PROGRAM MockServer
VAR
	//Mock Server
	fbhttpClient : FB_IotHttpClient := (sHostName:='4446f140-18dd-4b14-8279-3cc341a02b1e.mock.pstmn.io',
								  	bKeepAlive:=TRUE, tConnectionTimeout:=T#10S);		
				
	//Get Request
	fbRequest : FB_IotHttpRequest;		
	state : (IDLE, SEND_REQUEST, WAIT_FOR_RESPONSE, READ_RESPONSE,ERROR,HEADER);			
	sendGetRequest: BOOL;
	debugContent : STRING(511);
	fbJsonParser : FB_JsonDomParser;
	jsonDoc				: SJsonValue;
	jsonArgsMember				: SJsonValue;
	jsonMachineName : SJsonValue;
	results : STRING;
	
	//Header
	fbHeaderField : FB_IotHttpHeaderFieldMap;
END_VAR

// Init client parameters at startup
IF NOT fbhttpClient.bConfigured THEN 
	fbhttpClient.nHostPort:= 443; //80 for http  443 For https
	fbhttpClient.stTLS.bNoServerCertCheck:= TRUE;
END_IF

	
//Get Request
CASE state OF
	
	//Send Get Request
	IDLE:
		IF sendGetRequest THEN
			state := HEADER;
			sendGetRequest := FALSE;
		END_IF
	
	//Create Autorization Header File
	HEADER:
		fbHeaderField.AddField(sField:='Header1',sValue:='1',bAppendValue:=FALSE);
		fbHeaderField.AddField(sField:='Header2',sValue:='2',bAppendValue:=FALSE);
		state := SEND_REQUEST;
	
	//Send Get Request
	SEND_REQUEST:                                                                                      
		IF fbRequest.SendRequest(sUri:='/getmockdata', 
			fbClient:=fbhttpClient, eRequestType:=ETcIotHttpRequestType.HTTP_Get, 
				0, 0,fbHeader:=fbHeaderField ) THEN
			state := WAIT_FOR_RESPONSE;
		END_IF
	
	//Wait for Response
	WAIT_FOR_RESPONSE:

		IF NOT fbRequest.bBusy THEN
			IF fbRequest.bError THEN
				state := ERROR;
			ELSE
				state := READ_RESPONSE;
			END_IF
		END_IF
	
	//Read Response	
	READ_RESPONSE:
	
		//Get Response Content
		fbRequest.GetContent(pContent:= ADR(debugContent), nContentSize:= SIZEOF(debugContent), bSetNullTermination:= TRUE);
		
		//Check Status 
		IF fbRequest.nStatusCode >= 200 AND fbRequest.nStatusCode < 300 THEN
			jsonDoc:= fbRequest.GetJsonDomContent(fbJsonParser);
			
			//Check response has data in body
			IF jsonDoc <> 0 THEN
				
				//Check machine key is present 
				IF fbJsonParser.HasMember(jsonDoc, 'machine') THEN
					
					//Get Value for the specifed key
					jsonArgsMember:= fbJsonParser.FindMember(jsonDoc, 'machine');
					
					//Check wether data has an name key 	
					IF fbJsonParser.HasMember(jsonArgsMember, 'name')  THEN
						
						//Get Value for the specifed key
						jsonMachineName:= fbJsonParser.FindMember(jsonArgsMember, 'name');
						
							//Check data is a String
							IF fbJsonParser.IsString(jsonMachineName) THEN	
								
								//Get the Data 		
								results:= fbJsonParser.GetString(jsonMachineName);									
							END_IF
					END_IF
				END_IF
			END_IF
		END_IF
		state := IDLE;
		
	ERROR:
		//
		
		
END_CASE

//Cyclic Client 
fbhttpClient.Execute();

END_PROGRAM

(* stored: Version 1.1.0.1, ProductVersion 3.1.4024.12
   POU MockServer: Id {b95df168-f5ce-4f3b-b8ce-14883b6dc7b8}, SpecialFunc None *)
